// TIA Portal V17 export
// export: Created 2024-08-07T21:44:15.9032068Z, ExportSetting WithDefaults, DisplayName Totally Integrated Automation Portal, DisplayVersion V17 Update 7, DisplayName TIA Portal Openness, DisplayVersion V17 Update 7, DisplayName TIA Portal Version Control Interface, DisplayVersion V17, DisplayName SINAMICS Startdrive Advanced, DisplayVersion V17 SP2, DisplayName SINAMICS Startdrive G110M, G120, G120C, G120D, G120P, G115D, DisplayVersion V17 SP2, DisplayName SINAMICS Startdrive G130, G150, S120, S150, SINAMICS MV, S210, DisplayVersion V17 SP2, DisplayName STEP 7 Professional, DisplayVersion V17 Update 7, DisplayName STEP 7 Safety, DisplayVersion V17 Update 6, DisplayName WinCC Advanced / Unified PC, DisplayVersion V17 Update 7
TYPE "UDT_ProductionProgramProductCounters"
// stored: IsFailsafeCompliant false
   STRUCT
      Shift { S7_SetPoint := 'True'} : Array[1..3] of "UDT_Counters";
      Overall { S7_SetPoint := 'True'} : "UDT_Counters";
   END_STRUCT;
END_TYPE
